// TwinCAT 3 PLC project TcoKukaRobotics
// Title: TcoKukaRobotics
// Company: Vortex.Library
// Author: TcOpenGroup
// ProjectVersion: 0.6.0.913
// ProgramVersion: 3.1.4024.12
// libraries:
//   Tc2_MC2, * (Beckhoff Automation GmbH)
//   Tc2_MC2_Drive, * (Beckhoff Automation GmbH)
//   Tc2_Standard, * (Beckhoff Automation GmbH)
//   Tc2_System, * (Beckhoff Automation GmbH)
//   Tc3_Module, * (Beckhoff Automation GmbH)
//   TcoAbstractions, 0.6.0.913 (Vortex.Library)
//   TcoCore, 0.6.0.913 (Vortex.Library)
//   TcoIo, 0.6.0.913 (Vortex.Library)
//   TcoUtilities, 0.6.0.913 (Vortex.Library)
// project tree:
//   DUTs/ TcoKukaRobotics_Config_v_5_x_x.TcDUT (not stored), TcoKukaRobotics_Control_v_5_x_x.TcDUT (not stored), TcoKukaRobotics_State_v_5_x_x.TcDUT (not stored), TcoKukaRobotics_Status_v_5_x_x.TcDUT (not stored)
//   / PlcTask.TcTTO (not stored)
//   POUs/ MAIN.TcPOU (not stored)
//   POUs/Prototypes/KRC4/IO/ TcoKrc4_Inputs_v_5_x_x.TcDUT (not stored), TcoKrc4_IO_v_5_x_x.TcDUT (not stored), TcoKrc4_Outputs_v_5_x_x.TcDUT (not stored)
//   POUs/Prototypes/KRC4/ TcoKrc4_v_5_x_x.TcPOU, TcoKrc4_Ecat_v_5_x_x.TcPOU
//   POUs/Prototypes/RoboticsTasks/Starts/ StartAtMainTask.TcPOU (not stored), StartMotorsAndProgramTask.TcPOU, StartMotorsProgramAndMovementsTask.TcPOU (not stored), StartMotorsTask.TcPOU (not stored), StartMovementsTask.TcPOU (not stored), StartProgramTask.TcPOU
//   POUs/Prototypes/RoboticsTasks/Stops/ StopMotorsTask.TcPOU (not stored), StopMovementsAndProgramTask.TcPOU (not stored), StopMovementsTask.TcPOU (not stored), StopProgramTask.TcPOU (not stored)
//   POUs/Prototypes/RoboticsTasks/ TcoKukaRoboticsTask.TcPOU (not stored)

// ---- POUs/Prototypes/KRC4/TcoKrc4_v_5_x_x.TcPOU
FUNCTION_BLOCK TcoKrc4_v_5_x_x EXTENDS TcoIo.TcoPnIoComponent  IMPLEMENTS TcoAbstractions.ITcoRobotics
VAR_INPUT
    inEnable : BOOL;
END_VAR
VAR_OUTPUT
END_VAR
VAR_IN_OUT
    inoData : TcoKrc4_IO_v_5_x_x;
END_VAR
VAR
    

	{attribute addProperty Name "<#Status#>"}
    {attribute clr [ReadOnly()]}
    _status : TcoKukaRobotics_Status_v_5_x_x;
	{attribute addProperty Name "<#Control#>"}
	_control 	: TcoKukaRobotics_Control_v_5_x_x;
	{attribute addProperty Name "<#Config#>"}
    _config : TcoKukaRobotics_Config_v_5_x_x;
	{attribute addProperty Name "<#PN Error#>"}
    {attribute clr [ReadOnly()]}
    _busError : BOOL;
	//~
	_someTaskIsActive: BOOL;

	_stopTasksAreActive: BOOL;
	//~
	_reportTimer:TON;
END_VAR
VAR
	{attribute addProperty Name "<#Start at Main#>"}
    _startAtMainTask : StartAtMainTask(THIS^);
	
	 {attribute addProperty Name "<#Start motors and program#>"}
    _startMotorsAndProgramTask : StartMotorsAndProgramTask(THIS^);
	
	 {attribute addProperty Name "<#Start program#>"}
    _startProgramTask : StartProgramTask(THIS^);
	
	{attribute addProperty Name "<#Start motors#>"}
    _startMotorsTask : StartMotorsTask(THIS^);
	
  	{attribute addProperty Name "<#Start movements#>"}
    _startMovementsTask : StartMovementsTask(THIS^);
	
	{attribute addProperty Name "<#Start motors program and movements#>"}
    _startMotorsProgramAndMovementsTask : StartMotorsProgramAndMovementsTask(THIS^);
	
  	
	
	
	 {attribute addProperty Name "<#Stop movements#>"}
    _stopMovementsTask : StopMovementsTask(THIS^);

	 {attribute addProperty Name "<#Stop movenents and program#>"}
    _stopMovementsAndProgramTask : StopMovementsAndProgramTask(THIS^);
	
	{attribute addProperty Name "<#Stop program#>"}
    _stopProgramTask : StopProgramTask(THIS^);
	
	{attribute addProperty Name "<#Stop motors#>"}
    _stopMotorsTask : StopMotorsTask(THIS^);
	

    {attribute addProperty Name "<#Restore#>"}
    _restoreTask : TcoCore.TcoTask(THIS^);
	

  
   

  

END_VAR

VAR
	{attribute 'hide'}
	_sb : TcoCore.StringBuilder;
END_VAR

IF NOT __ISVALIDREF(inoData) THEN
    Messenger.Post('Invalid reference', TcoCore.eMessageCategory.ProgrammingError);
    RETURN;
END_IF

SUPER^(inPnIoBoxState := THIS^.inoData.PnIoBoxState, inPnIoBoxDiag := THIS^.inoData.PnIoBoxDiag);
_busError := NOT _profinetReady;

UpdateStatus();
_stopTasksAreActive := _stopMovementsTask.Busy AND _stopMovementsAndProgramTask.Busy AND _stopProgramTask.Busy AND _stopMotorsTask.Busy;

_startAtMainTask.Enabled := NOT _stopTasksAreActive;
_startAtMainTask(inoConfig := _config, inoControl := _control, inoStatus := _status);

_startProgramTask.Enabled := NOT _stopTasksAreActive;
_startProgramTask(inoConfig := _config, inoControl := _control, inoStatus := _status);

_startMotorsTask.Enabled := NOT _stopTasksAreActive AND NOT _startMotorsProgramAndMovementsTask.Busy AND NOT _startMotorsAndProgramTask.Busy;
_startMotorsTask(inoConfig := _config, inoControl := _control, inoStatus := _status);

_startMotorsAndProgramTask.Enabled := NOT _stopTasksAreActive AND NOT _startProgramTask.Busy AND NOT _startMotorsTask.Busy;
_startMotorsAndProgramTask(inoConfig := _config, inoControl := _control, inoStatus := _status);

_startMovementsTask.Enabled := NOT _startMotorsProgramAndMovementsTask.Busy AND NOT _stopMotorsTask.Busy;
_startMovementsTask(inoConfig := _config, inoControl := _control, inoStatus := _status);

_startMotorsProgramAndMovementsTask.Enabled := NOT _startMovementsTask.Busy AND NOT _stopMotorsTask.Busy;
_startMotorsProgramAndMovementsTask(refStartMotorsAndProgramTask := _startMotorsAndProgramTask,
    inoConfig := _config,
    inoControl := _control,
    inoStatus := _status);

_stopMovementsTask.Enabled := TRUE;
_stopMovementsTask(inoConfig := _config, inoControl := _control, inoStatus := _status);

_stopMotorsTask.Enabled := TRUE;
_stopMotorsTask(inoConfig := _config, inoControl := _control, inoStatus := _status);

_stopProgramTask.Enabled := TRUE;
_stopProgramTask(inoConfig := _config, inoControl := _control, inoStatus := _status);

_stopMovementsAndProgramTask.Enabled := NOT _stopProgramTask.Busy AND NOT _stopProgramTask.Busy;
_stopMovementsAndProgramTask(inoConfig := _config, inoControl := _control, inoStatus := _status);

//*************RESTORE********************

_restoreTask.Enabled := TRUE;

IF _restoreTask.Execute() THEN
    Restore();
    _restoreTask.DoneWhen(TRUE);
END_IF

//****************************************

_someTaskIsActive := _startAtMainTask.Busy OR
    _startMotorsAndProgramTask.Busy OR
    _startMovementsTask.Busy OR
    _startMovementsTask.Busy OR
    _stopMovementsTask.Busy OR
    _stopMovementsAndProgramTask.Busy OR
    _stopProgramTask.Busy;

//do not publish diagnostic message when component is not used
IF _someTaskIsActive THEN

    IF (NOT _status.State.AlarmStopActive) THEN
        Messenger.Error('<#Emergency stop active#>');
    END_IF;

    IF (NOT _status.State.UserSafetySwitchClosed) THEN
        Messenger.Warning('<#Safety Error #>');
    END_IF;

END_IF;

_reportTimer(IN := Status.State.Manual AND NOT Status.State.Automatic, PT := _config.InfoTime);

Messenger.OnCondition(_reportTimer.Q AND _status.State.Error).Error(_sb.Clear()
        .Append('<#Robot reported an error: #>')
        .Append(UDINT_TO_STRING(_status.State.EventId))
        .Append(' |[[0]AdvancedDiagnosticMessage]|')
        .Append('.')
        .Append('For details see the service mode')
        .ToString());

IF Status.State.Manual AND NOT Status.State.Automatic THEN
    _control.MoveEnable := TRUE; //robotic department request
    Messenger.OnCondition(_reportTimer.Q).Warning(_sb.Clear().Append('<#Robot in Maual. MoveEnable is Forced!#>').ToString());
END_IF

UpdateControl();

(*~
	<docu>
		<summary>
			Gets the configuration of the IRC 5. 					
		</summary>			
	</docu>	
~*)
PROPERTY Config : REFERENCE TO TcoKukaRobotics_Config_v_5_x_x
GET
Config REF= _config;
END_GET
END_PROPERTY

PROPERTY PUBLIC Control : REFERENCE TO TcoKukaRobotics_Control_v_5_x_x
GET
Control REF= _control;
END_GET
END_PROPERTY

METHOD FB_init : BOOL
VAR_INPUT
	bInitRetains : BOOL; // if TRUE, the retain variables are initialized (warm start / cold start)
	bInCopyCode : BOOL;  // if TRUE, the instance afterwards gets moved into the copy code (online change)
  	ParentObject : ITcoObject;	
END_VAR
END_METHOD

(*~
	<docu>
		<summary>
			Restores this instance to the Ready state. Can be called explicitly or from within one of the restore mechanisms.	
		</summary>			
	</docu>	
~*)
METHOD Restore : ITcoRestorable
RestoreTasks();

_control.GlobalSpeed:=0;
_control.ActivateInterface:=FALSE;
_control.ErrorConfirmation:=FALSE;
_control.ExternalStart:=FALSE;

_control.MasterMode:=0;


//todo to restore control signals
_control.ToolNo:=0;
_control.WorkobjectNo:=0;
_control.PointNo:=0;
_control.UserSpecSpeed1:=0;
_control.UserSpecSpeed2:=0;
_control.Coordinates.X:=0;
_control.Coordinates.Y:=0;
_control.Coordinates.Z:=0;
_control.Coordinates.Rx:=0;
_control.Coordinates.Ry:=0;
_control.Coordinates.Rz:=0;
END_METHOD

METHOD INTERNAL RestoreTasks
//_resetTask.Restore();
_startAtMainTask.Restore();
_startMovementsTask.Restore();
_startProgramTask.Restore();
_startMotorsTask.Restore();
_stopMotorsTask.Restore();
_startMotorsProgramAndMovementsTask.Restore();
_stopMovementsTask.Restore();
_startMotorsAndProgramTask.Restore();
_stopMovementsAndProgramTask.Restore();
_stopProgramTask.Restore();
END_METHOD

(*~
	<docu>
		<summary>
		    Custom service (manual, maintenance) logic.
			This method must be implemented in derived class.
		</summary>			
	</docu>	
~*)
METHOD PROTECTED ServiceMode
END_METHOD

METHOD PUBLIC StartAtMain : TcoCore.ITcoTaskStatus
VAR_INPUT
END_VAR
StartAtMain:=_startAtMainTask.Invoke();
END_METHOD

PROPERTY StartAtMainTask : TcoCore.ITcoTaskStatus
GET
StartAtMainTask := _startAtMainTask;
END_GET
END_PROPERTY

METHOD PUBLIC StartMotors : TcoCore.ITcoTaskStatus
StartMotors:=_startMotorsTask.Invoke();
END_METHOD

METHOD StartMotorsAndProgram : TcoCore.ITcoTaskStatus
VAR_INPUT
END_VAR
StartMotorsAndProgram := THIS^._startMotorsAndProgramTask.Invoke();
END_METHOD

PROPERTY StartMotorsAndProgramTask : TcoCore.ITcoTaskStatus
GET
StartMotorsAndProgramTask := _startMotorsAndProgramTask;
END_GET
END_PROPERTY

METHOD PUBLIC StartMotorsProgramAndMovements : TcoCore.ITcoTaskStatus
VAR_INPUT
	inData : TcoRoboticsMovementsParams;
END_VAR
StartMotorsProgramAndMovements:=_startMotorsProgramAndMovementsTask.InvokeWithParams(inData);
END_METHOD

PROPERTY StartMotorsProgramAndMovementsTask : TcoCore.ITcoTaskStatus
GET
StartMotorsProgramAndMovementsTask := _startMotorsProgramAndMovementsTask;
END_GET
END_PROPERTY

PROPERTY StartMotorsTask : TcoCore.ITcoTaskStatus
GET
StartMotorsTask := _startMotorsTask;
END_GET
END_PROPERTY

METHOD PUBLIC StartMovements : TcoCore.ITcoTaskStatus
VAR_INPUT
	inData : TcoRoboticsMovementsParams;
END_VAR
StartMovements:=_startMovementsTask.InvokeWithParams(inData);
END_METHOD

PROPERTY StartMovementsTask : TcoCore.ITcoTaskStatus
GET
StartMovementsTask := _startMovementsTask;
END_GET
END_PROPERTY

METHOD PUBLIC StartProgram : TcoCore.ITcoTaskStatus
StartProgram:=_startProgramTask.Invoke();
END_METHOD

PROPERTY StartProgramTask : TcoCore.ITcoTaskStatus
GET
StartProgramTask := _startProgramTask;
END_GET
END_PROPERTY

(*~
	<docu>
		<summary>
			Gets the status of the IRC5. 					
		</summary>			
	</docu>	
~*)
PROPERTY Status : REFERENCE TO TcoKukaRobotics_Status_v_5_x_x
GET
Status REF= _status;
END_GET
END_PROPERTY

METHOD PUBLIC StopMotors : TcoCore.ITcoTaskStatus
StopMotors:=_stopMotorsTask.Invoke();
END_METHOD

PROPERTY StopMotorsTask : TcoCore.ITcoTaskStatus
GET
StopMotorsTask := _stopMotorsTask;
END_GET
END_PROPERTY

METHOD PUBLIC StopMovements : TcoCore.ITcoTaskStatus
VAR_INPUT
	inStopType : eTcoRoboticsStopType;
END_VAR
StopMovements:=_stopMovementsTask.InvokeWithParams(inStopType);
END_METHOD

METHOD PUBLIC StopMovementsAndProgram : TcoCore.ITcoTaskStatus
VAR_INPUT
	inStopType : eTcoRoboticsStopType;
END_VAR
StopMovementsAndProgram:=_stopMovementsAndProgramTask.InvokeWithParams(inStopType);
END_METHOD

PROPERTY StopMovementsAndProgramTask : TcoCore.ITcoTaskStatus
GET
StopMovementsAndProgramTask := _stopMovementsAndProgramTask;
END_GET
END_PROPERTY

PROPERTY StopMovementsTask : TcoCore.ITcoTaskStatus
GET
StopMovementsTask := _stopMovementsTask;
END_GET
END_PROPERTY

METHOD PUBLIC StopProgram : TcoCore.ITcoTaskStatus
StopProgram:=_stopProgramTask.Invoke();
END_METHOD

PROPERTY StopProgramTask : TcoCore.ITcoTaskStatus
GET
StopProgramTask := _stopProgramTask;
END_GET
END_PROPERTY

METHOD INTERNAL UpdateControl
VAR_INPUT
END_VAR

VAR
	index: INT;
END_VAR
//SYSTEM OUTPUTS
index:=0;
inoData.Out.Outputs[index].0	:=		_control.ExternalStart;    
inoData.Out.Outputs[index].1	:=		_control.MoveEnable;    
inoData.Out.Outputs[index].2 	:= 		_control.ErrorConfirmation; 
inoData.Out.Outputs[index].3 	:= 		_control.DrivesOff;
inoData.Out.Outputs[index].4 	:= 		_control.DrivesOn;   
inoData.Out.Outputs[index].5 	:= 		_control.ActivateInterface; 
inoData.Out.Outputs[index].6 	:= 		_control.StartAtMain;    


//index:=1;
//inoData.Out.Outputs[index].0 	:= 		_control.StartProgram;    
//inoData.Out.Outputs[index].1 	:= 		_control.StartAtMain;    
//inoData.Out.Outputs[index].2 	:= 		_control.StopProgram;    
//inoData.Out.Outputs[index].3 	:= 		_control.QuickStop;    
//inoData.Out.Outputs[index].4 	:= 		_control.SoftStop;    
//inoData.Out.Outputs[index].5 	:= 		_control.StopCycle;    
//inoData.Out.Outputs[index].6 	:= 		_control.StopInstruction;    
//inoData.Out.Outputs[index].7 	:= 		_control.LimitSpeed;    


	
//Tool signals
index:=2;
inoData.Out.Outputs[index].0 	:= 		_control.Tool_1_Retract;    
inoData.Out.Outputs[index].1 	:= 		_control.Tool_1_Extend;    
inoData.Out.Outputs[index].2	:= 		_control.Tool_2_Retract;    
inoData.Out.Outputs[index].3	:= 		_control.Tool_2_Extend;    
inoData.Out.Outputs[index].4	:= 		_control.Tool_3_Retract;    
inoData.Out.Outputs[index].5	:= 		_control.Tool_3_Extend;    
inoData.Out.Outputs[index].6 	:= 		_control.Tool_4_Retract;    
inoData.Out.Outputs[index].7	:= 		_control.Tool_4_Extend;    
//master mode  such as manual/auto ....
index:=3;
inoData.Out.Outputs[index]:= _control.MasterMode;
//zone
index:=5;
inoData.Out.Outputs[index]:= _control.Zone;
//position
index:=6;
inoData.Out.Outputs[index]:= _control.InPosition;

//
//Movement parameters
index:=7;
inoData.Out.Outputs[index]:= _control.ActionNo;
index:=8;
inoData.Out.Outputs[index]:= _control.GlobalSpeed;
index:=9;
inoData.Out.Outputs[index]:= _control.ToolNo;
index:=10;
inoData.Out.Outputs[index]:= _control.WorkobjectNo;
index:=11;
inoData.Out.Outputs[index]:= _control.PointNo;
index:=12;
TcoUtilities.TcoDintToBytes(inFormat:=TcoUtilities.eTcoDataFormat.LittleEndian,
							inValue:=REAL_TO_DINT(_control.UserSpecSpeed1),
							outByte0:=inoData.Out.Outputs[index],
							outByte1:=inoData.Out.Outputs[index+1],
							outByte2:=inoData.Out.Outputs[index+2],
							outByte3:=inoData.Out.Outputs[index+3]);
index:=16;
TcoUtilities.TcoDintToBytes(inFormat:=TcoUtilities.eTcoDataFormat.LittleEndian,
							inValue:=REAL_TO_DINT(_control.UserSpecSpeed2),
							outByte0:=inoData.Out.Outputs[index],
							outByte1:=inoData.Out.Outputs[index+1],
							outByte2:=inoData.Out.Outputs[index+2],
							outByte3:=inoData.Out.Outputs[index+3]);

////Coordinates
index:=20;
TcoUtilities.TcoDintToBytes(inFormat:=TcoUtilities.eTcoDataFormat.LittleEndian,
							inValue:=REAL_TO_DINT((_control.Coordinates.X)*10000.0),
							outByte0:=inoData.Out.Outputs[index],
							outByte1:=inoData.Out.Outputs[index+1],
							outByte2:=inoData.Out.Outputs[index+2],
							outByte3:=inoData.Out.Outputs[index+3]);
index:=24;
TcoUtilities.TcoDintToBytes(inFormat:=TcoUtilities.eTcoDataFormat.LittleEndian,
							inValue:=REAL_TO_DINT((_control.Coordinates.Y)*10000.0),
							outByte0:=inoData.Out.Outputs[index],
							outByte1:=inoData.Out.Outputs[index+1],
							outByte2:=inoData.Out.Outputs[index+2],
							outByte3:=inoData.Out.Outputs[index+3]);
index:=28;
TcoUtilities.TcoDintToBytes(inFormat:=TcoUtilities.eTcoDataFormat.LittleEndian,
							inValue:=REAL_TO_DINT((_control.Coordinates.Z)*10000.0),
							outByte0:=inoData.Out.Outputs[index],
							outByte1:=inoData.Out.Outputs[index+1],
							outByte2:=inoData.Out.Outputs[index+2],
							outByte3:=inoData.Out.Outputs[index+3]);
index:=32;
TcoUtilities.TcoDintToBytes(inFormat:=TcoUtilities.eTcoDataFormat.LittleEndian,
							inValue:=REAL_TO_DINT((_control.Coordinates.Rx)*10000.0),
							outByte0:=inoData.Out.Outputs[index],
							outByte1:=inoData.Out.Outputs[index+1],
							outByte2:=inoData.Out.Outputs[index+2],
							outByte3:=inoData.Out.Outputs[index+3]);
index:=36;
TcoUtilities.TcoDintToBytes(inFormat:=TcoUtilities.eTcoDataFormat.LittleEndian,
							inValue:=REAL_TO_DINT((_control.Coordinates.Ry)*10000.0),
							outByte0:=inoData.Out.Outputs[index],
							outByte1:=inoData.Out.Outputs[index+1],
							outByte2:=inoData.Out.Outputs[index+2],
							outByte3:=inoData.Out.Outputs[index+3]);
index:=40;
TcoUtilities.TcoDintToBytes(inFormat:=TcoUtilities.eTcoDataFormat.LittleEndian,
							inValue:=REAL_TO_DINT((_control.Coordinates.Rz)*10000.0),
							outByte0:=inoData.Out.Outputs[index],
							outByte1:=inoData.Out.Outputs[index+1],
							outByte2:=inoData.Out.Outputs[index+2],
							outByte3:=inoData.Out.Outputs[index+3]);
END_METHOD

METHOD INTERNAL UpdateStatus
VAR
    _message : STRING(125);

	tempOut: BYTE;
	index: INT;
	_bytes: DINT;
END_VAR
//SYSTEM INPUTS
index:=0;
_status.State.RcReady := inoData.In.Inputs[index].0;
_status.State.AlarmStopActive := inoData.In.Inputs[index].1;
_status.State.UserSafetySwitchClosed := inoData.In.Inputs[index].2;
_status.State.DrivesReady := inoData.In.Inputs[index].3;
_status.State.RobotCalibrated := inoData.In.Inputs[index].4;
_status.State.InterfaceActivated := inoData.In.Inputs[index].5;
_status.State.StopMess := inoData.In.Inputs[index].6;
_status.State.RobotStopped := inoData.In.Inputs[index].7;

index:=1;
_status.State.InHome := inoData.In.Inputs[index].0;
_status.State.Manual := inoData.In.Inputs[index].1;
_status.State.Automatic := inoData.In.Inputs[index].2;
_status.State.ExternalAutomatic := inoData.In.Inputs[index].3;
_status.State.ProActive := inoData.In.Inputs[index].4;
_status.State.PpMoved := inoData.In.Inputs[index].5;
_status.State.Error := inoData.In.Inputs[index].6;
_status.State.ProgramMoveActive := inoData.In.Inputs[index].7;


//Area/positions flags this  should be obsolete because Zones and InPosition is used as byte below
index:=2;
_status.State.InArea_1 := inoData.In.Inputs[index].0;
_status.State.InArea_2 := inoData.In.Inputs[index].1;
_status.State.InArea_3 := inoData.In.Inputs[index].2;
_status.State.InArea_4 := inoData.In.Inputs[index].3;
_status.State.InPosition_1 := inoData.In.Inputs[index].4;
_status.State.InPosition_2 := inoData.In.Inputs[index].5;
_status.State.InPosition_3 := inoData.In.Inputs[index].6;
_status.State.InPosition_4 := inoData.In.Inputs[index].7;
//
//Tool signals
index:=3;
_status.State.Tool_1_Retract := inoData.In.Inputs[index].0;
_status.State.Tool_1_Extend := inoData.In.Inputs[index].1;
_status.State.Tool_2_Retract := inoData.In.Inputs[index].2;
_status.State.Tool_2_Extend := inoData.In.Inputs[index].3;
_status.State.Tool_3_Retract := inoData.In.Inputs[index].4;
_status.State.Tool_3_Extend := inoData.In.Inputs[index].5;
_status.State.Tool_4_Retract := inoData.In.Inputs[index].6;
_status.State.Tool_4_Extend := inoData.In.Inputs[index].7;

//Safety signals
index:=4;


index:=5;
_status.State.Zone:= inoData.In.Inputs[index];
index:=6;
_status.State.InPosition:= inoData.In.Inputs[index];

//Movement parameters
index:=7;
_status.State.ActionNo:= inoData.In.Inputs[index];
index:=8;
_status.State.GlobalSpeed:= inoData.In.Inputs[index];
index:=9;
_status.State.ToolNo:= inoData.In.Inputs[index];
index:=10;
_status.State.WorkobjectNo:= inoData.In.Inputs[index];
index:=11;
_status.State.PointNo:= inoData.In.Inputs[index];
index:=12;
_status.State.UserSpecSpeed1:=TcoUtilities.TcoBytesToDint (inFormat:=TcoUtilities.eTcoDataFormat.LittleEndian,
															inByte0:= inoData.In.Inputs[index],
															inByte1:= inoData.In.Inputs[index+1],
															inByte2:= inoData.In.Inputs[index+2],
															inByte3:= inoData.In.Inputs[index+3]);
index:=16;
_status.State.UserSpecSpeed2:=TcoUtilities.TcoBytesToDint (inFormat:=TcoUtilities.eTcoDataFormat.LittleEndian,
															inByte0:= inoData.In.Inputs[index],
															inByte1:= inoData.In.Inputs[index+1],
															inByte2:= inoData.In.Inputs[index+2],
															inByte3:= inoData.In.Inputs[index+3]);
															
index:=20;
_bytes:=TcoUtilities.TcoBytesToDint (inFormat:=TcoUtilities.eTcoDataFormat.LittleEndian,
															inByte0:= inoData.In.Inputs[index],
															inByte1:= inoData.In.Inputs[index+1],
															inByte2:= inoData.In.Inputs[index+2],
															inByte3:= inoData.In.Inputs[index+3]);

_status.State.Coordinates.X:=(DINT_TO_REAL(_bytes)/10000.0);

index:=24;
_bytes:=TcoUtilities.TcoBytesToDint (inFormat:=TcoUtilities.eTcoDataFormat.LittleEndian,
															inByte0:= inoData.In.Inputs[index],
															inByte1:= inoData.In.Inputs[index+1],
															inByte2:= inoData.In.Inputs[index+2],
															inByte3:= inoData.In.Inputs[index+3]);

_status.State.Coordinates.Y:=(DINT_TO_REAL(_bytes)/10000.0);

index:=28;
_bytes:=TcoUtilities.TcoBytesToDint (inFormat:=TcoUtilities.eTcoDataFormat.LittleEndian,
															inByte0:= inoData.In.Inputs[index],
															inByte1:= inoData.In.Inputs[index+1],
															inByte2:= inoData.In.Inputs[index+2],
															inByte3:= inoData.In.Inputs[index+3]);

_status.State.Coordinates.Z:=(DINT_TO_REAL(_bytes)/10000.0);

index:=32;															
_bytes:=TcoUtilities.TcoBytesToDint (inFormat:=TcoUtilities.eTcoDataFormat.LittleEndian,
															inByte0:= inoData.In.Inputs[index],
															inByte1:= inoData.In.Inputs[index+1],
															inByte2:= inoData.In.Inputs[index+2],
															inByte3:= inoData.In.Inputs[index+3]);

_status.State.Coordinates.Rx:=(DINT_TO_REAL(_bytes)/10000.0);

index:=36;
_bytes:=TcoUtilities.TcoBytesToDint (inFormat:=TcoUtilities.eTcoDataFormat.LittleEndian,
															inByte0:= inoData.In.Inputs[index],
															inByte1:= inoData.In.Inputs[index+1],
															inByte2:= inoData.In.Inputs[index+2],
															inByte3:= inoData.In.Inputs[index+3]);

_status.State.Coordinates.Ry:=(DINT_TO_REAL(_bytes)/10000.0);

index:=40;
_bytes:=TcoUtilities.TcoBytesToDint (inFormat:=TcoUtilities.eTcoDataFormat.LittleEndian,
															inByte0:= inoData.In.Inputs[index],
															inByte1:= inoData.In.Inputs[index+1],
															inByte2:= inoData.In.Inputs[index+2],
															inByte3:= inoData.In.Inputs[index+3]);

_status.State.Coordinates.Rz:=(DINT_TO_REAL(_bytes)/10000.0);

index:=44;
_status.State.EventId:=TcoUtilities.TcoBytesToUDint (inFormat:=TcoUtilities.eTcoDataFormat.LittleEndian,
															inByte0:= inoData.In.Inputs[index],
															inByte1:= inoData.In.Inputs[index+1],
															inByte2:= inoData.In.Inputs[index+2],
															inByte3:= inoData.In.Inputs[index+3]);
END_METHOD

END_FUNCTION_BLOCK

// ---- POUs/Prototypes/RoboticsTasks/Starts/StartMotorsAndProgramTask.TcPOU
FUNCTION_BLOCK StartMotorsAndProgramTask EXTENDS TcoKukaRoboticsTask



IF Execute() THEN
	 _blink(inOnTime:=T#500MS,inOffTime:=T#500MS);

  	IF _progress = 0 THEN
		IF NOT __ISVALIDREF(inoControl) THEN
			_varInfo :=__VARINFO(inoControl);
			Messenger.Programming(_sb.Clear().Append('<#Invalid reference: #>').Append(_varInfo.Symbol).ToString()).Pin();
		ELSIF NOT __ISVALIDREF(inoConfig) THEN                                                  
			_varInfo :=__VARINFO(inoConfig);                                                    
			Messenger.Programming(_sb.Clear().Append('<#Invalid reference: #>').Append(_varInfo.Symbol).ToString()).Pin();
		ELSIF NOT __ISVALIDREF(inoStatus) THEN                                                  
			_varInfo :=__VARINFO(inoStatus);                                                    
			Messenger.Programming(_sb.Clear().Append('<#Invalid reference: #>').Append(_varInfo.Symbol).ToString()).Pin();
		ELSE

			_progress := _progress + 1;

		END_IF

	END_IF
	IF _progress = 1 THEN
	
		_varInfo :=__VARINFO( inoStatus.State.UserSafetySwitchClosed);                                                
		THIS^.Messenger.OnCondition(_infoTimer.Q AND NOT inoStatus.State.UserSafetySwitchClosed).Warning(_sb.Clear().Append('<#Waiting for signal#>').Append(_varInfo.Symbol).ToString());
		IF  inoStatus.State.UserSafetySwitchClosed THEN
			_progress := _progress + 1;
		END_IF;
	END_IF;
	IF _progress = 2 THEN
	
		_varInfo :=__VARINFO( inoStatus.State.AlarmStopActive);                                                
		THIS^.Messenger.OnCondition(_infoTimer.Q AND NOT inoStatus.State.AlarmStopActive).Warning(_sb.Clear().Append('<#Waiting for signal#>').Append(_varInfo.Symbol).ToString());
		IF  inoStatus.State.AlarmStopActive THEN
			_progress := _progress + 1;
		END_IF;
	END_IF;

	IF _progress = 3 THEN	

		_varInfo :=__VARINFO( inoStatus.State.DrivesReady);                                                
		THIS^.Messenger.OnCondition(_infoTimer.Q AND NOT inoStatus.State.DrivesReady).Warning(_sb.Clear().Append('<# Waiting for signal: #>').Append(_varInfo.Symbol).ToString());
		inoControl.DrivesOff:=TRUE;		
		inoControl.DrivesOn:=_blink.outQ;	
		IF inoStatus.State.DrivesReady  THEN
			 inoControl.DrivesOn:=FALSE;
			_progress := _progress + 1;
		END_IF
	END_IF;		
	
	
	IF _progress = 4 THEN	
		Messenger.Debug('<#Robot Error Reset and Move Enable#>');
		
		inoControl.ErrorConfirmation := inoStatus.State.StopMess AND _blink.outQ;
		_varInfo :=__VARINFO( inoStatus.State.StopMess);                                                
		THIS^.Messenger.OnCondition(_infoTimer.Q AND  inoStatus.State.StopMess).Warning(_sb.Clear().Append('<#Waiting for signal#>').Append(_varInfo.Symbol).Append(' is OFF').ToString());

		_varInfo :=__VARINFO( inoStatus.State.RcReady);                                                
		THIS^.Messenger.OnCondition(_infoTimer.Q AND NOT inoStatus.State.RcReady).Warning(_sb.Clear().Append('<#Waiting for signal#>').Append(_varInfo.Symbol).ToString());

		IF NOT inoStatus.State.StopMess AND inoStatus.State.RcReady THEN
			inoControl.ErrorConfirmation:=FALSE;
			_progress := _progress + 1;
		END_IF
	END_IF;
	
	IF _progress = 5 THEN
	
		inoControl.ActivateInterface:=TRUE;
		_varInfo :=__VARINFO( inoStatus.State.InterfaceActivated);                                                
		THIS^.Messenger.OnCondition(_infoTimer.Q AND NOT inoStatus.State.InterfaceActivated).Warning(_sb.Clear().Append('<#Waiting for signal#>').Append(_varInfo.Symbol).ToString());
		IF  inoStatus.State.InterfaceActivated THEN
			_progress := _progress + 1;
		END_IF;
	END_IF;
	
	IF _progress = 6 THEN	
		IF inoStatus.State.StopMess OR inoStatus.State.AlarmStopActive OR NOT  inoStatus.State.RcReady THEN 
			_progress := 1;
		END_IF
		inoControl.ExternalStart:=_blink.outQ;
		_varInfo :=__VARINFO( inoStatus.State.ProActive);                                                
		THIS^.Messenger.OnCondition(_infoTimer.Q AND NOT inoStatus.State.ProActive).Warning(_sb.Clear().Append('<#Waiting for program running signal! #>').Append(_varInfo.Symbol).ToString());
		
		
		IF  inoStatus.State.ProActive  THEN
				inoControl.ExternalStart:=FALSE;
		END_IF
	END_IF;
	
    DoneWhen(inoStatus.State.ProActive AND inoStatus.State.DrivesReady AND NOT inoStatus.State.StopMess);
    CallTimers(TRUE);
	THIS^.ThrowWhen(_errorTimer.Q );
	
END_IF

IF  THIS^.Error AND NOT _errorMessage.Pinned THEN
	THIS^.Restore();
END_IF

METHOD PUBLIC FB_init : BOOL
VAR_INPUT
    bInitRetains : BOOL; // if TRUE, the retain variables are initialized (warm start / cold start)
    bInCopyCode : BOOL; // if TRUE, the instance afterwards gets moved into the copy code (online change)
    ParentObject : ITcoObject;	
END_VAR
END_METHOD

(*~
	<docu>
		<summary>
			Executes when task is aborted.
		</summary>			
	</docu>	
~*)
METHOD PROTECTED OnAbort
IF  __ISVALIDREF(inoStatus) THEN   THIS^.inoStatus.ActionDescription := '<#Start motors and program was aborted.#>'; END_IF;
inoControl.MoveEnable := false;
END_METHOD

(*~
	<docu>
		<summary>
			Executes when task reaches the ```Done``` state .
		</summary>			
	</docu>	
~*)
METHOD PROTECTED OnDone
IF  __ISVALIDREF(inoStatus) THEN   THIS^.inoStatus.ActionDescription := '<#Start motors and program finished successfully.#>'; END_IF;
_progress:=0;
inoControl.ActivateInterface:=FALSE;
END_METHOD

METHOD PROTECTED OnError

VAR
	description: STRING;
END_VAR
description := '<#Start motors and program finished with error.#>'; 
IF  __ISVALIDREF(inoStatus) THEN   THIS^.inoStatus.ActionDescription := description; END_IF;
THIS^._errorMessage.Error(_sb.Clear().Append(description).Append(' To restore acknowledge this alarm.').ToString()).Pin();
END_METHOD

METHOD PROTECTED OnStart
IF  __ISVALIDREF(inoStatus) THEN  THIS^.inoStatus.ActionDescription := '<#Start motors and program started.#>'; END_IF; 
CallTimers(FALSE);
inoControl.MoveEnable := TRUE;
END_METHOD

(*~
	<docu>
		<summary>
			Restores this instance to the Ready state. Can be called explicitly or from within one of the restore mechanisms.
			<para>
				See also <see cref="PlcDocu.TcoCore.TcoTask.AutoRestorable()"/>
			</para>
		</summary>			
	</docu>	
~*)
METHOD Restore : ITcoRestorable
SUPER^.Restore();
END_METHOD

END_FUNCTION_BLOCK

// ---- POUs/Prototypes/RoboticsTasks/Starts/StartProgramTask.TcPOU
FUNCTION_BLOCK StartProgramTask EXTENDS TcoKukaRoboticsTask
VAR

	_stopType: TcoAbstractions.eTcoRoboticsStopType;
END_VAR



IF Execute() THEN
	_blink(inOnTime:=T#500MS,inOffTime:=T#500MS);

	IF _progress = 0 THEN
		IF NOT __ISVALIDREF(inoControl) THEN
			_varInfo :=__VARINFO(inoControl);
			Messenger.Programming(_sb.Clear().Append('<#Invalid reference: #>').Append(_varInfo.Symbol).ToString()).Pin();
		ELSIF NOT __ISVALIDREF(inoConfig) THEN                                                  
			_varInfo :=__VARINFO(inoConfig);                                                    
			Messenger.Programming(_sb.Clear().Append('<#Invalid reference: #>').Append(_varInfo.Symbol).ToString()).Pin();
		ELSIF NOT __ISVALIDREF(inoStatus) THEN                                                  
			_varInfo :=__VARINFO(inoStatus);                                                    
			Messenger.Programming(_sb.Clear().Append('<#Invalid reference: #>').Append(_varInfo.Symbol).ToString()).Pin();
			ELSE
			_progress := _progress + 1;
		END_IF

	END_IF
		
	
	
	
	IF _progress = 1 THEN
	
		_varInfo :=__VARINFO( inoStatus.State.UserSafetySwitchClosed);                                                
		THIS^.Messenger.OnCondition(_infoTimer.Q AND NOT inoStatus.State.UserSafetySwitchClosed).Warning(_sb.Clear().Append('<#Waiting for signal#>').Append(_varInfo.Symbol).ToString());
		IF  inoStatus.State.UserSafetySwitchClosed THEN
			_progress := _progress + 1;
		END_IF;
	END_IF;
	IF _progress = 2 THEN
	
		_varInfo :=__VARINFO( inoStatus.State.AlarmStopActive);                                                
		THIS^.Messenger.OnCondition(_infoTimer.Q AND NOT inoStatus.State.AlarmStopActive).Warning(_sb.Clear().Append('<#Waiting for signal#>').Append(_varInfo.Symbol).ToString());
		IF  inoStatus.State.AlarmStopActive THEN
			_progress := _progress + 1;
		END_IF;
	END_IF;

	IF _progress = 3 THEN	

		_varInfo :=__VARINFO( inoStatus.State.DrivesReady);                                                
		THIS^.Messenger.OnCondition(_infoTimer.Q AND NOT inoStatus.State.DrivesReady).Warning(_sb.Clear().Append('<# Waiting for signal: #>').Append(_varInfo.Symbol).ToString());
		inoControl.DrivesOff:=TRUE;		
		inoControl.DrivesOn:=_blink.outQ;	
		IF inoStatus.State.DrivesReady  THEN
			 inoControl.DrivesOn:=FALSE;
			_progress := _progress + 1;
		END_IF
	END_IF;		
	
	
	IF _progress = 4 THEN	
		Messenger.Debug('<#Robot Error Reset and Move Enable#>');
	
		inoControl.ErrorConfirmation := inoStatus.State.StopMess AND _blink.outQ;
		_varInfo :=__VARINFO( inoStatus.State.StopMess);                                                
		THIS^.Messenger.OnCondition(_infoTimer.Q AND  inoStatus.State.StopMess).Warning(_sb.Clear().Append('<#Waiting for signal#>').Append(_varInfo.Symbol).Append(' is OFF').ToString());

		_varInfo :=__VARINFO( inoStatus.State.RcReady);                                                
		THIS^.Messenger.OnCondition(_infoTimer.Q AND NOT inoStatus.State.RcReady).Warning(_sb.Clear().Append('<#Waiting for signal#>').Append(_varInfo.Symbol).ToString());

		IF NOT inoStatus.State.StopMess AND inoStatus.State.RcReady THEN
			inoControl.ErrorConfirmation:=FALSE;
			_progress := _progress + 1;
		END_IF
	END_IF;
	
	IF _progress = 5 THEN
	
		inoControl.ActivateInterface:=TRUE;
		_varInfo :=__VARINFO( inoStatus.State.InterfaceActivated);                                                
		THIS^.Messenger.OnCondition(_infoTimer.Q AND NOT inoStatus.State.InterfaceActivated).Warning(_sb.Clear().Append('<#Waiting for signal#>').Append(_varInfo.Symbol).ToString());
		IF  inoStatus.State.InterfaceActivated THEN
			_progress := _progress + 1;
		END_IF;
	END_IF;
	
	IF _progress = 6 THEN	
		IF inoStatus.State.StopMess OR inoStatus.State.AlarmStopActive OR NOT  inoStatus.State.RcReady THEN 
			_progress := 1;
		END_IF
		inoControl.ExternalStart:=_blink.outQ;
		_varInfo :=__VARINFO( inoStatus.State.ProActive);                                                
		THIS^.Messenger.OnCondition(_infoTimer.Q AND NOT inoStatus.State.ProActive).Warning(_sb.Clear().Append('<#Waiting for program running signal! #>').Append(_varInfo.Symbol).ToString());
		
		
		IF  inoStatus.State.ProActive  THEN
				inoControl.ExternalStart:=FALSE;
		END_IF
	END_IF;		
	
	
    DoneWhen(inoStatus.State.ProActive AND inoStatus.State.DrivesReady AND NOT inoStatus.State.StopMess);
    CallTimers(TRUE);
	
	THIS^.ThrowWhen(_errorTimer.Q );
END_IF

IF  THIS^.Error AND NOT _errorMessage.Pinned THEN
	THIS^.Restore();
END_IF

METHOD PUBLIC FB_init : BOOL
VAR_INPUT
    bInitRetains : BOOL; // if TRUE, the retain variables are initialized (warm start / cold start)
    bInCopyCode : BOOL; // if TRUE, the instance afterwards gets moved into the copy code (online change)
  	ParentObject : ITcoObject;	
END_VAR
END_METHOD

METHOD INTERNAL InvokeWithParams : ITcoTaskStatus
VAR_INPUT
	inStopType : eTcoRoboticsStopType;
END_VAR
_stopType := inStopType;
InvokeWithParams := THIS^.Invoke();
END_METHOD

(*~
	<docu>
		<summary>
			Executes when task is aborted.
		</summary>			
	</docu>	
~*)
METHOD PROTECTED OnAbort
IF  __ISVALIDREF(inoStatus) THEN   THIS^.inoStatus.ActionDescription := '<#Start program was aborted, while not yet completed!#>';END_IF; 
inoControl.MoveEnable := FALSE;
END_METHOD

(*~
	<docu>
		<summary>
			Executes when task reaches the ```Done``` state .
		</summary>			
	</docu>	
~*)
METHOD PROTECTED OnDone
IF  __ISVALIDREF(inoStatus) THEN  THIS^.inoStatus.ActionDescription := '<#Stop program was completed successfully.#>';END_IF; 
_progress:=0;
inoControl.ActivateInterface:=FALSE;
END_METHOD

(*~
	<docu>
		<summary>
			Executes when task reaches the ```Error``` state.
				</summary>			
	</docu>	
~*)
METHOD PROTECTED OnError
VAR
	description: STRING;
END_VAR
THIS^.inoStatus.ActionDescription := '<#Stopping program with error.#>'; 
IF  __ISVALIDREF(inoStatus) THEN   THIS^.inoStatus.ActionDescription := description; END_IF;
THIS^._errorMessage.Error(_sb.Clear().Append(description).Append(' To restore acknowledge this alarm.').ToString()).Pin();
END_METHOD

METHOD PROTECTED OnStart
IF  __ISVALIDREF(inoStatus) THEN  THIS^.inoStatus.ActionDescription := '<#Starting program started.#>'; END_IF; 
CallTimers(FALSE);
inoControl.MoveEnable:=TRUE;
END_METHOD

(*~
	<docu>
		<summary>
			Restores this instance to the Ready state. Can be called explicitly or from within one of the restore mechanisms.
			<para>
				See also <see cref="PlcDocu.TcoCore.TcoTask.AutoRestorable()"/>
			</para>
		</summary>			
	</docu>	
~*)
METHOD Restore : ITcoRestorable
SUPER^.Restore();
END_METHOD

END_FUNCTION_BLOCK

// ---- POUs/Prototypes/KRC4/TcoKrc4_Ecat_v_5_x_x.TcPOU
FUNCTION_BLOCK TcoKrc4_Ecat_v_5_x_x EXTENDS TcoIo.TcoEcatComponent  IMPLEMENTS TcoAbstractions.ITcoRobotics
VAR_INPUT
    inEnable : BOOL;
END_VAR
VAR_OUTPUT
END_VAR
VAR_IN_OUT
    inoData : TcoKrc4_IO_v_5_x_x;
END_VAR
VAR
    

	{attribute addProperty Name "<#Status#>"}
    {attribute clr [ReadOnly()]}
    _status : TcoKukaRobotics_Status_v_5_x_x;
	{attribute addProperty Name "<#Control#>"}
	_control 	: TcoKukaRobotics_Control_v_5_x_x;
	{attribute addProperty Name "<#Config#>"}
    _config : TcoKukaRobotics_Config_v_5_x_x;
	{attribute addProperty Name "<#ECat Error#>"}
    {attribute clr [ReadOnly()]}
    _busError : BOOL;

	_someTaskIsActive: BOOL;

	_stopTasksAreActive: BOOL;
END_VAR
VAR
	{attribute addProperty Name "<#Start at Main#>"}
    _startAtMainTask : StartAtMainTask(THIS^);
	
	 {attribute addProperty Name "<#Start motors and program#>"}
    _startMotorsAndProgramTask : StartMotorsAndProgramTask(THIS^);
	
	 {attribute addProperty Name "<#Start program#>"}
    _startProgramTask : StartProgramTask(THIS^);
	
	{attribute addProperty Name "<#Start motors#>"}
    _startMotorsTask : StartMotorsTask(THIS^);
	
  	{attribute addProperty Name "<#Start movements#>"}
    _startMovementsTask : StartMovementsTask(THIS^);
	
	{attribute addProperty Name "<#Start motors program and movements#>"}
    _startMotorsProgramAndMovementsTask : StartMotorsProgramAndMovementsTask(THIS^);
	
  	
	
	
	 {attribute addProperty Name "<#Stop movements#>"}
    _stopMovementsTask : StopMovementsTask(THIS^);

	 {attribute addProperty Name "<#Stop movenents and program#>"}
    _stopMovementsAndProgramTask : StopMovementsAndProgramTask(THIS^);
	
	{attribute addProperty Name "<#Stop program#>"}
    _stopProgramTask : StopProgramTask(THIS^);
	
	{attribute addProperty Name "<#Stop motors#>"}
    _stopMotorsTask : StopMotorsTask(THIS^);
	

    {attribute addProperty Name "<#Restore#>"}
    _restoreTask : TcoCore.TcoTask(THIS^);
	

  
   

  

END_VAR

IF NOT __ISVALIDREF(inoData) THEN
    Messenger.Post('Invalid reference', TcoCore.eMessageCategory.ProgrammingError);
    RETURN;
END_IF

SUPER^(AdsAddr:=AdsAddr);
_busError:= NOT SUPER^._ecatState.EcatOk;



UpdateStatus();
_stopTasksAreActive :=  _stopMovementsTask.Busy 
			AND _stopMovementsAndProgramTask.Busy 
			AND _stopProgramTask.Busy
			AND _stopMotorsTask.Busy;
			
_startAtMainTask.Enabled:=NOT _stopTasksAreActive;
_startAtMainTask(inoConfig:=_config,inoControl:=_control,inoStatus:=_status);


_startProgramTask.Enabled:=NOT _stopTasksAreActive;
_startProgramTask(inoConfig:=_config,inoControl:=_control,inoStatus:=_status);

_startMotorsTask.Enabled:=NOT _stopTasksAreActive AND NOT _startMotorsProgramAndMovementsTask.Busy AND NOT _startMotorsAndProgramTask.Busy;
_startMotorsTask(inoConfig:=_config,inoControl:=_control,inoStatus:=_status);

_startMotorsAndProgramTask.Enabled:=NOT _stopTasksAreActive AND NOT _startProgramTask.Busy AND NOT _startMotorsTask.Busy;
_startMotorsAndProgramTask(inoConfig:=_config,inoControl:=_control,inoStatus:=_status);

_startMovementsTask.Enabled:=NOT _startMotorsProgramAndMovementsTask.Busy AND NOT _stopMotorsTask.Busy;
_startMovementsTask(inoConfig:=_config,inoControl:=_control,inoStatus:=_status);

_startMotorsProgramAndMovementsTask.Enabled:=NOT _startMovementsTask.Busy  AND NOT _stopMotorsTask.Busy;
_startMotorsProgramAndMovementsTask(refStartMotorsAndProgramTask:=_startMotorsAndProgramTask, inoConfig:=_config,inoControl:=_control,inoStatus:=_status);


_stopMovementsTask.Enabled:=TRUE;
_stopMovementsTask(inoConfig:=_config,inoControl:=_control,inoStatus:=_status);

_stopMotorsTask.Enabled:=TRUE;
_stopMotorsTask(inoConfig:=_config,inoControl:=_control,inoStatus:=_status);

_stopProgramTask.Enabled:=TRUE;
_stopProgramTask(inoConfig:=_config,inoControl:=_control,inoStatus:=_status);

_stopMovementsAndProgramTask.Enabled:=NOT _stopProgramTask.Busy AND NOT _stopProgramTask.Busy;
_stopMovementsAndProgramTask(inoConfig:=_config,inoControl:=_control,inoStatus:=_status);



//*************RESTORE********************

_restoreTask.Enabled := TRUE;
IF _restoreTask.Execute() THEN
	Restore();
	_restoreTask.DoneWhen(TRUE);
END_IF
//****************************************

_someTaskIsActive := _startAtMainTask.Busy 
					OR _startMotorsAndProgramTask.Busy
					OR _startMovementsTask.Busy
					OR _startMovementsTask.Busy
					OR _stopMovementsTask.Busy
					OR _stopMovementsAndProgramTask.Busy
					OR _stopProgramTask.Busy;
					

//do not publish diagnostic message when component is not used
IF _someTaskIsActive THEN

	IF(NOT _status.State.AlarmStopActive) THEN
		Messenger.Error('<#Emergency stop active#>');
	END_IF;
	IF(NOT _status.State.UserSafetySwitchClosed) THEN
		Messenger.Warning('<#Safety Error #>');
	END_IF;

  
END_IF;


IF(_status.State.Error) THEN Messenger.Error(_sb.Clear().Append('<#Robot reported an error: #>').Append(UDINT_TO_STRING(_status.State.EventId)).Append(' |[[0]AdvancedDiagnosticMessage]|').Append('.').Append('For details see the service mode').ToString()); END_IF;


UpdateControl();

(*~
	<docu>
		<summary>
			Gets the configuration of the IRC 5. 					
		</summary>			
	</docu>	
~*)
PROPERTY Config : REFERENCE TO TcoKukaRobotics_Config_v_5_x_x
GET
Config REF= _config;
END_GET
END_PROPERTY

PROPERTY PUBLIC Control : REFERENCE TO TcoKukaRobotics_Control_v_5_x_x
GET
Control REF= _control;
END_GET
END_PROPERTY

METHOD FB_init : BOOL
VAR_INPUT
	bInitRetains : BOOL; // if TRUE, the retain variables are initialized (warm start / cold start)
	bInCopyCode : BOOL;  // if TRUE, the instance afterwards gets moved into the copy code (online change)
  	ParentObject : ITcoObject;	
END_VAR
END_METHOD

(*~
	<docu>
		<summary>
			Restores this instance to the Ready state. Can be called explicitly or from within one of the restore mechanisms.	
		</summary>			
	</docu>	
~*)
METHOD Restore : ITcoRestorable
RestoreTasks();

_control.GlobalSpeed:=0;
_control.ActivateInterface:=FALSE;
_control.ErrorConfirmation:=FALSE;
_control.ExternalStart:=FALSE;

_control.MasterMode:=0;


//todo to restore control signals
_control.ToolNo:=0;
_control.WorkobjectNo:=0;
_control.PointNo:=0;
_control.UserSpecSpeed1:=0;
_control.UserSpecSpeed2:=0;
_control.Coordinates.X:=0;
_control.Coordinates.Y:=0;
_control.Coordinates.Z:=0;
_control.Coordinates.Rx:=0;
_control.Coordinates.Ry:=0;
_control.Coordinates.Rz:=0;
END_METHOD

METHOD INTERNAL RestoreTasks
//_resetTask.Restore();
_startAtMainTask.Restore();
_startMovementsTask.Restore();
_startProgramTask.Restore();
_startMotorsTask.Restore();
_stopMotorsTask.Restore();
_startMotorsProgramAndMovementsTask.Restore();
_stopMovementsTask.Restore();
_startMotorsAndProgramTask.Restore();
_stopMovementsAndProgramTask.Restore();
_stopProgramTask.Restore();
END_METHOD

(*~
	<docu>
		<summary>
		    Custom service (manual, maintenance) logic.
			This method must be implemented in derived class.
		</summary>			
	</docu>	
~*)
METHOD PROTECTED ServiceMode
END_METHOD

METHOD PUBLIC StartAtMain : TcoCore.ITcoTaskStatus
VAR_INPUT
END_VAR
StartAtMain:=_startAtMainTask.Invoke();
END_METHOD

PROPERTY StartAtMainTask : TcoCore.ITcoTaskStatus
GET
StartAtMainTask := _startAtMainTask;
END_GET
END_PROPERTY

METHOD PUBLIC StartMotors : TcoCore.ITcoTaskStatus
StartMotors:=_startMotorsTask.Invoke();
END_METHOD

METHOD StartMotorsAndProgram : TcoCore.ITcoTaskStatus
VAR_INPUT
END_VAR
StartMotorsAndProgram := THIS^._startMotorsAndProgramTask.Invoke();
END_METHOD

PROPERTY StartMotorsAndProgramTask : TcoCore.ITcoTaskStatus
GET
StartMotorsAndProgramTask := _startMotorsAndProgramTask;
END_GET
END_PROPERTY

METHOD PUBLIC StartMotorsProgramAndMovements : TcoCore.ITcoTaskStatus
VAR_INPUT
	inData : TcoRoboticsMovementsParams;
END_VAR
StartMotorsProgramAndMovements:=_startMotorsProgramAndMovementsTask.InvokeWithParams(inData);
END_METHOD

PROPERTY StartMotorsProgramAndMovementsTask : TcoCore.ITcoTaskStatus
GET
StartMotorsProgramAndMovementsTask := _startMotorsProgramAndMovementsTask;
END_GET
END_PROPERTY

PROPERTY StartMotorsTask : TcoCore.ITcoTaskStatus
GET
StartMotorsTask := _startMotorsTask;
END_GET
END_PROPERTY

METHOD PUBLIC StartMovements : TcoCore.ITcoTaskStatus
VAR_INPUT
	inData : TcoRoboticsMovementsParams;
END_VAR
StartMovements:=_startMovementsTask.InvokeWithParams(inData);
END_METHOD

PROPERTY StartMovementsTask : TcoCore.ITcoTaskStatus
GET
StartMovementsTask := _startMovementsTask;
END_GET
END_PROPERTY

METHOD PUBLIC StartProgram : TcoCore.ITcoTaskStatus
StartProgram:=_startProgramTask.Invoke();
END_METHOD

PROPERTY StartProgramTask : TcoCore.ITcoTaskStatus
GET
StartProgramTask := _startProgramTask;
END_GET
END_PROPERTY

(*~
	<docu>
		<summary>
			Gets the status of the IRC5. 					
		</summary>			
	</docu>	
~*)
PROPERTY Status : REFERENCE TO TcoKukaRobotics_Status_v_5_x_x
GET
Status REF= _status;
END_GET
END_PROPERTY

METHOD PUBLIC StopMotors : TcoCore.ITcoTaskStatus
StopMotors:=_stopMotorsTask.Invoke();
END_METHOD

PROPERTY StopMotorsTask : TcoCore.ITcoTaskStatus
GET
StopMotorsTask := _stopMotorsTask;
END_GET
END_PROPERTY

METHOD PUBLIC StopMovements : TcoCore.ITcoTaskStatus
VAR_INPUT
	inStopType : eTcoRoboticsStopType;
END_VAR
StopMovements:=_stopMovementsTask.InvokeWithParams(inStopType);
END_METHOD

METHOD PUBLIC StopMovementsAndProgram : TcoCore.ITcoTaskStatus
VAR_INPUT
	inStopType : eTcoRoboticsStopType;
END_VAR
StopMovementsAndProgram:=_stopMovementsAndProgramTask.InvokeWithParams(inStopType);
END_METHOD

PROPERTY StopMovementsAndProgramTask : TcoCore.ITcoTaskStatus
GET
StopMovementsAndProgramTask := _stopMovementsAndProgramTask;
END_GET
END_PROPERTY

PROPERTY StopMovementsTask : TcoCore.ITcoTaskStatus
GET
StopMovementsTask := _stopMovementsTask;
END_GET
END_PROPERTY

METHOD PUBLIC StopProgram : TcoCore.ITcoTaskStatus
StopProgram:=_stopProgramTask.Invoke();
END_METHOD

PROPERTY StopProgramTask : TcoCore.ITcoTaskStatus
GET
StopProgramTask := _stopProgramTask;
END_GET
END_PROPERTY

METHOD INTERNAL UpdateControl
VAR_INPUT
END_VAR

VAR
	index: INT;
END_VAR
//SYSTEM OUTPUTS
index:=0;
inoData.Out.Outputs[index].0	:=		_control.ExternalStart;    
inoData.Out.Outputs[index].1	:=		_control.MoveEnable;    
inoData.Out.Outputs[index].2 	:= 		_control.ErrorConfirmation; 
inoData.Out.Outputs[index].3 	:= 		_control.DrivesOff;
inoData.Out.Outputs[index].4 	:= 		_control.DrivesOn;   
inoData.Out.Outputs[index].5 	:= 		_control.ActivateInterface; 
inoData.Out.Outputs[index].6 	:= 		_control.StartAtMain;    


//index:=1;
//inoData.Out.Outputs[index].0 	:= 		_control.StartProgram;    
//inoData.Out.Outputs[index].1 	:= 		_control.StartAtMain;    
//inoData.Out.Outputs[index].2 	:= 		_control.StopProgram;    
//inoData.Out.Outputs[index].3 	:= 		_control.QuickStop;    
//inoData.Out.Outputs[index].4 	:= 		_control.SoftStop;    
//inoData.Out.Outputs[index].5 	:= 		_control.StopCycle;    
//inoData.Out.Outputs[index].6 	:= 		_control.StopInstruction;    
//inoData.Out.Outputs[index].7 	:= 		_control.LimitSpeed;    


	
//Tool signals
index:=2;
inoData.Out.Outputs[index].0 	:= 		_control.Tool_1_Retract;    
inoData.Out.Outputs[index].1 	:= 		_control.Tool_1_Extend;    
inoData.Out.Outputs[index].2	:= 		_control.Tool_2_Retract;    
inoData.Out.Outputs[index].3	:= 		_control.Tool_2_Extend;    
inoData.Out.Outputs[index].4	:= 		_control.Tool_3_Retract;    
inoData.Out.Outputs[index].5	:= 		_control.Tool_3_Extend;    
inoData.Out.Outputs[index].6 	:= 		_control.Tool_4_Retract;    
inoData.Out.Outputs[index].7	:= 		_control.Tool_4_Extend;    
//master mode  such as manual/auto ....
index:=3;
inoData.Out.Outputs[index]:= _control.MasterMode;
//zone
index:=5;
inoData.Out.Outputs[index]:= _control.Zone;
//position
index:=6;
inoData.Out.Outputs[index]:= _control.InPosition;

//
//Movement parameters
index:=7;
inoData.Out.Outputs[index]:= _control.ActionNo;
index:=8;
inoData.Out.Outputs[index]:= _control.GlobalSpeed;
index:=9;
inoData.Out.Outputs[index]:= _control.ToolNo;
index:=10;
inoData.Out.Outputs[index]:= _control.WorkobjectNo;
index:=11;
inoData.Out.Outputs[index]:= _control.PointNo;
index:=12;
TcoUtilities.TcoDintToBytes(inFormat:=TcoUtilities.eTcoDataFormat.LittleEndian,
							inValue:=REAL_TO_DINT(_control.UserSpecSpeed1),
							outByte0:=inoData.Out.Outputs[index],
							outByte1:=inoData.Out.Outputs[index+1],
							outByte2:=inoData.Out.Outputs[index+2],
							outByte3:=inoData.Out.Outputs[index+3]);
index:=16;
TcoUtilities.TcoDintToBytes(inFormat:=TcoUtilities.eTcoDataFormat.LittleEndian,
							inValue:=REAL_TO_DINT(_control.UserSpecSpeed2),
							outByte0:=inoData.Out.Outputs[index],
							outByte1:=inoData.Out.Outputs[index+1],
							outByte2:=inoData.Out.Outputs[index+2],
							outByte3:=inoData.Out.Outputs[index+3]);

////Coordinates
index:=20;
TcoUtilities.TcoDintToBytes(inFormat:=TcoUtilities.eTcoDataFormat.LittleEndian,
							inValue:=REAL_TO_DINT((_control.Coordinates.X)*10000.0),
							outByte0:=inoData.Out.Outputs[index],
							outByte1:=inoData.Out.Outputs[index+1],
							outByte2:=inoData.Out.Outputs[index+2],
							outByte3:=inoData.Out.Outputs[index+3]);
index:=24;
TcoUtilities.TcoDintToBytes(inFormat:=TcoUtilities.eTcoDataFormat.LittleEndian,
							inValue:=REAL_TO_DINT((_control.Coordinates.Y)*10000.0),
							outByte0:=inoData.Out.Outputs[index],
							outByte1:=inoData.Out.Outputs[index+1],
							outByte2:=inoData.Out.Outputs[index+2],
							outByte3:=inoData.Out.Outputs[index+3]);
index:=28;
TcoUtilities.TcoDintToBytes(inFormat:=TcoUtilities.eTcoDataFormat.LittleEndian,
							inValue:=REAL_TO_DINT((_control.Coordinates.Z)*10000.0),
							outByte0:=inoData.Out.Outputs[index],
							outByte1:=inoData.Out.Outputs[index+1],
							outByte2:=inoData.Out.Outputs[index+2],
							outByte3:=inoData.Out.Outputs[index+3]);
index:=32;
TcoUtilities.TcoDintToBytes(inFormat:=TcoUtilities.eTcoDataFormat.LittleEndian,
							inValue:=REAL_TO_DINT((_control.Coordinates.Rx)*10000.0),
							outByte0:=inoData.Out.Outputs[index],
							outByte1:=inoData.Out.Outputs[index+1],
							outByte2:=inoData.Out.Outputs[index+2],
							outByte3:=inoData.Out.Outputs[index+3]);
index:=36;
TcoUtilities.TcoDintToBytes(inFormat:=TcoUtilities.eTcoDataFormat.LittleEndian,
							inValue:=REAL_TO_DINT((_control.Coordinates.Ry)*10000.0),
							outByte0:=inoData.Out.Outputs[index],
							outByte1:=inoData.Out.Outputs[index+1],
							outByte2:=inoData.Out.Outputs[index+2],
							outByte3:=inoData.Out.Outputs[index+3]);
index:=40;
TcoUtilities.TcoDintToBytes(inFormat:=TcoUtilities.eTcoDataFormat.LittleEndian,
							inValue:=REAL_TO_DINT((_control.Coordinates.Rz)*10000.0),
							outByte0:=inoData.Out.Outputs[index],
							outByte1:=inoData.Out.Outputs[index+1],
							outByte2:=inoData.Out.Outputs[index+2],
							outByte3:=inoData.Out.Outputs[index+3]);
END_METHOD

METHOD INTERNAL UpdateStatus
VAR
    _message : STRING(125);

	tempOut: BYTE;
	index: INT;
	_bytes: DINT;
END_VAR
//SYSTEM INPUTS
index:=0;
_status.State.RcReady := inoData.In.Inputs[index].0;
_status.State.AlarmStopActive := inoData.In.Inputs[index].1;
_status.State.UserSafetySwitchClosed := inoData.In.Inputs[index].2;
_status.State.DrivesReady := inoData.In.Inputs[index].3;
_status.State.RobotCalibrated := inoData.In.Inputs[index].4;
_status.State.InterfaceActivated := inoData.In.Inputs[index].5;
_status.State.StopMess := inoData.In.Inputs[index].6;
_status.State.RobotStopped := inoData.In.Inputs[index].7;

index:=1;
_status.State.InHome := inoData.In.Inputs[index].0;
_status.State.Manual := inoData.In.Inputs[index].1;
_status.State.Automatic := inoData.In.Inputs[index].2;
_status.State.ExternalAutomatic := inoData.In.Inputs[index].3;
_status.State.ProActive := inoData.In.Inputs[index].4;
_status.State.PpMoved := inoData.In.Inputs[index].5;
_status.State.Error := inoData.In.Inputs[index].6;
_status.State.ProgramMoveActive := inoData.In.Inputs[index].7;


//Area/positions flags this  should be obsolete because Zones and InPosition is used as byte below
index:=2;
_status.State.InArea_1 := inoData.In.Inputs[index].0;
_status.State.InArea_2 := inoData.In.Inputs[index].1;
_status.State.InArea_3 := inoData.In.Inputs[index].2;
_status.State.InArea_4 := inoData.In.Inputs[index].3;
_status.State.InPosition_1 := inoData.In.Inputs[index].4;
_status.State.InPosition_2 := inoData.In.Inputs[index].5;
_status.State.InPosition_3 := inoData.In.Inputs[index].6;
_status.State.InPosition_4 := inoData.In.Inputs[index].7;
//
//Tool signals
index:=3;
_status.State.Tool_1_Retract := inoData.In.Inputs[index].0;
_status.State.Tool_1_Extend := inoData.In.Inputs[index].1;
_status.State.Tool_2_Retract := inoData.In.Inputs[index].2;
_status.State.Tool_2_Extend := inoData.In.Inputs[index].3;
_status.State.Tool_3_Retract := inoData.In.Inputs[index].4;
_status.State.Tool_3_Extend := inoData.In.Inputs[index].5;
_status.State.Tool_4_Retract := inoData.In.Inputs[index].6;
_status.State.Tool_4_Extend := inoData.In.Inputs[index].7;

//Safety signals
index:=4;


index:=5;
_status.State.Zone:= inoData.In.Inputs[index];
index:=6;
_status.State.InPosition:= inoData.In.Inputs[index];

//Movement parameters
index:=7;
_status.State.ActionNo:= inoData.In.Inputs[index];
index:=8;
_status.State.GlobalSpeed:= inoData.In.Inputs[index];
index:=9;
_status.State.ToolNo:= inoData.In.Inputs[index];
index:=10;
_status.State.WorkobjectNo:= inoData.In.Inputs[index];
index:=11;
_status.State.PointNo:= inoData.In.Inputs[index];
index:=12;
_status.State.UserSpecSpeed1:=TcoUtilities.TcoBytesToDint (inFormat:=TcoUtilities.eTcoDataFormat.LittleEndian,
															inByte0:= inoData.In.Inputs[index],
															inByte1:= inoData.In.Inputs[index+1],
															inByte2:= inoData.In.Inputs[index+2],
															inByte3:= inoData.In.Inputs[index+3]);
index:=16;
_status.State.UserSpecSpeed2:=TcoUtilities.TcoBytesToDint (inFormat:=TcoUtilities.eTcoDataFormat.LittleEndian,
															inByte0:= inoData.In.Inputs[index],
															inByte1:= inoData.In.Inputs[index+1],
															inByte2:= inoData.In.Inputs[index+2],
															inByte3:= inoData.In.Inputs[index+3]);
															
index:=20;
_bytes:=TcoUtilities.TcoBytesToDint (inFormat:=TcoUtilities.eTcoDataFormat.LittleEndian,
															inByte0:= inoData.In.Inputs[index],
															inByte1:= inoData.In.Inputs[index+1],
															inByte2:= inoData.In.Inputs[index+2],
															inByte3:= inoData.In.Inputs[index+3]);

_status.State.Coordinates.X:=(DINT_TO_REAL(_bytes)/10000.0);

index:=24;
_bytes:=TcoUtilities.TcoBytesToDint (inFormat:=TcoUtilities.eTcoDataFormat.LittleEndian,
															inByte0:= inoData.In.Inputs[index],
															inByte1:= inoData.In.Inputs[index+1],
															inByte2:= inoData.In.Inputs[index+2],
															inByte3:= inoData.In.Inputs[index+3]);

_status.State.Coordinates.Y:=(DINT_TO_REAL(_bytes)/10000.0);

index:=28;
_bytes:=TcoUtilities.TcoBytesToDint (inFormat:=TcoUtilities.eTcoDataFormat.LittleEndian,
															inByte0:= inoData.In.Inputs[index],
															inByte1:= inoData.In.Inputs[index+1],
															inByte2:= inoData.In.Inputs[index+2],
															inByte3:= inoData.In.Inputs[index+3]);

_status.State.Coordinates.Z:=(DINT_TO_REAL(_bytes)/10000.0);

index:=32;															
_bytes:=TcoUtilities.TcoBytesToDint (inFormat:=TcoUtilities.eTcoDataFormat.LittleEndian,
															inByte0:= inoData.In.Inputs[index],
															inByte1:= inoData.In.Inputs[index+1],
															inByte2:= inoData.In.Inputs[index+2],
															inByte3:= inoData.In.Inputs[index+3]);

_status.State.Coordinates.Rx:=(DINT_TO_REAL(_bytes)/10000.0);

index:=36;
_bytes:=TcoUtilities.TcoBytesToDint (inFormat:=TcoUtilities.eTcoDataFormat.LittleEndian,
															inByte0:= inoData.In.Inputs[index],
															inByte1:= inoData.In.Inputs[index+1],
															inByte2:= inoData.In.Inputs[index+2],
															inByte3:= inoData.In.Inputs[index+3]);

_status.State.Coordinates.Ry:=(DINT_TO_REAL(_bytes)/10000.0);

index:=40;
_bytes:=TcoUtilities.TcoBytesToDint (inFormat:=TcoUtilities.eTcoDataFormat.LittleEndian,
															inByte0:= inoData.In.Inputs[index],
															inByte1:= inoData.In.Inputs[index+1],
															inByte2:= inoData.In.Inputs[index+2],
															inByte3:= inoData.In.Inputs[index+3]);

_status.State.Coordinates.Rz:=(DINT_TO_REAL(_bytes)/10000.0);

index:=44;
_status.State.EventId:=TcoUtilities.TcoBytesToUDint (inFormat:=TcoUtilities.eTcoDataFormat.LittleEndian,
															inByte0:= inoData.In.Inputs[index],
															inByte1:= inoData.In.Inputs[index+1],
															inByte2:= inoData.In.Inputs[index+2],
															inByte3:= inoData.In.Inputs[index+3]);
END_METHOD

END_FUNCTION_BLOCK
